FUNCTION_BLOCK CAT1_Motion (* Composite Function Block Type *)
  (* Standard: 61499-2 *)
  (* Version 0.0, 2/19/2024, SESA658662, Schneider Electric, template *)
  PACKAGE Main;
  {SET_ATTRIBUTE(AllowExtendableInterface, 1)}
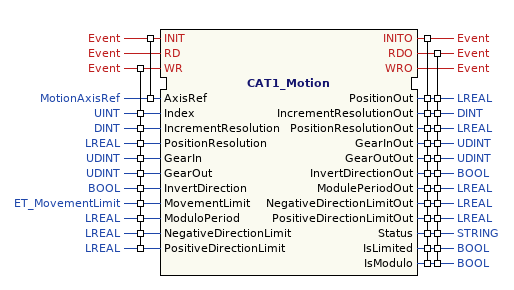
  EVENT_INPUT
    INIT WITH AxisRef; (* Service Request *)
    RD;
    WR WITH IncrementResolution, PositionResolution, GearIn, GearOut, InvertDirection, Index, ModuloPeriod, NegativeDirectionLimit, PositiveDirectionLimit, MovementLimit; (* Service Request *)
  END_EVENT
  EVENT_OUTPUT
    INITO WITH PositionOut, IncrementResolutionOut, PositionResolutionOut, GearInOut, GearOutOut, InvertDirectionOut, Status, ModulePeriodOut, NegativeDirectionLimitOut, PositiveDirectionLimitOut, IsLimited, IsModulo;
    RDO WITH PositionOut, IncrementResolutionOut, PositionResolutionOut, GearInOut, GearOutOut, InvertDirectionOut, Status, ModulePeriodOut, NegativeDirectionLimitOut, PositiveDirectionLimitOut, IsLimited, IsModulo; (* Confirmation of Requested Service *)
    WRO;
  END_EVENT
  VAR_INPUT
    AxisRef : MotionAxisRef;
    Index : UINT;
    IncrementResolution : DINT;
    PositionResolution : LREAL;
    GearIn : UDINT;
    GearOut : UDINT;
    InvertDirection : BOOL;
    MovementLimit : ET_MovementLimit;
    ModuloPeriod : LREAL;
    NegativeDirectionLimit : LREAL;
    PositiveDirectionLimit : LREAL;
  END_VAR
  VAR_OUTPUT
    PositionOut : LREAL;
    IncrementResolutionOut : DINT;
    PositionResolutionOut : LREAL;
    GearInOut : UDINT;
    GearOutOut : UDINT;
    InvertDirectionOut : BOOL;
    ModulePeriodOut : LREAL;
    NegativeDirectionLimitOut : LREAL;
    PositiveDirectionLimitOut : LREAL;
    Status : STRING;
    IsLimited : BOOL;
    IsModulo : BOOL;
  END_VAR
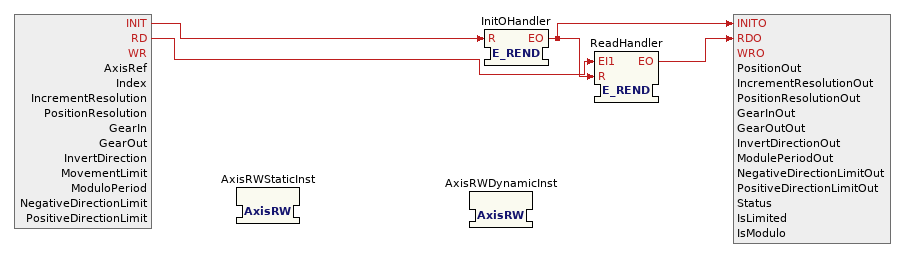
  (* Placeholder for initialising logic axis parameters with constant values *)
  (* Placeholder for writing logix axis parameters dynamically *)
  FBS
    AxisRWStaticInst : AxisRW;
    AxisRWDynamicInst : AxisRW;
    InitOHandler : E_REND;
    ReadHandler : E_REND;
  END_FBS
  EVENT_CONNECTIONS
    ReadHandler.EO TO RDO;
    InitOHandler.EO TO INITO;
    INIT TO InitOHandler.R;
    RD TO ReadHandler.EI1;
    InitOHandler.EO TO ReadHandler.R;
  END_CONNECTIONS
END_FUNCTION_BLOCK
